{attribute addProperty BoxType "KL2300-0100"}
{attribute addProperty Id "InputAT %I*BOOL000OutputAT %Q*BOOL000"}
{attribute addProperty CRC "3090566181"}
{attribute addProperty SizeInBites "0"}
{attribute addProperty SizeInBytes "0"}
TYPE Channel_B8364C25 :
STRUCT
	{attribute addProperty Name "Input"}
	Input AT %I* : BOOL;
	{attribute addProperty Name "Output"}
	Output AT %Q* : BOOL;
END_STRUCT
END_TYPE

(* stored: Version 1.2.0.0, ProductVersion 3.1.4024.9
   DUT Channel_B8364C25: Id {9a7cb476-3ce7-45cf-a324-6fa71675c10d} *)
